FUNCTION_BLOCK StackerCraneProcess
VAR_IN_OUT
	bStart : BOOL;
	bHalt : BOOL;
	bResume : BOOL;
	bStop : BOOL;
	fioOutputs : OUTPUTS;
END_VAR
VAR_INPUT
	fioInputs : INPUTS;
	iAlgo: INT;
	iMode: INT;
	iRackSlot : INT;
END_VAR
VAR_OUTPUT
	sCurrentOperation : STRING;
	iTotalPalletsProcessed : INT;
	iPalletsInRack : INT;
	aSlots : ARRAY[1..54] OF BOOL;

END_VAR
VAR
	bFirstStart : BOOL := TRUE;
	
	iStep : INT := 0;
	bPalletWaiting : BOOL;
	startTrig : R_TRIG;
	stopTrig : R_TRIG;
	resumeTrig : R_TRIG;
	haltTrig : R_TRIG;
	iHaltStep : INT;
	mAlgo : INT;
	mMode : INT;
	i : INT;
	iChosenSlot : INT;
	fill : Fill;
	empty : Empty;
	home : Home;
	iCounter :INT;
	exitTimer : TON;
	infoTimer : TON;
	aFillVerticalPositions : ARRAY[1..54] OF INT := [
		1, 10, 19, 28, 37, 46,
		2, 11, 20, 29, 38, 47,
		3, 12, 21, 30, 39, 48,
		4, 13, 22, 31, 40, 49,
		5, 14, 23, 32, 41, 50,
		6, 15, 24, 33, 42, 51,
		7, 16, 25, 34, 43, 52,
		8, 17, 26, 35, 44, 53,
		9, 18, 27, 36, 45, 54
	];
	
	aEmptyVerticalPositions : ARRAY[1..54] OF INT := [
		54, 45, 36, 27, 18, 9,
		53, 44, 35, 26, 17, 8,
		52, 43, 34, 25, 16, 7,
		51, 42, 33, 24, 15, 6,
		50, 41, 32, 23, 14, 5,
		49, 40, 31, 22, 13, 4,
		48, 39, 30, 21, 12, 3,
		47, 38, 29, 20, 11, 2,
		46, 37, 28, 19, 10, 1
	];
	storedOutputs : OUTPUTS;
	haltedOutputs : OUTPUTS;
	sStoredCurrentOp : STRING;
	
END_VAR

VAR CONSTANT
	AVAILABLE_SLOTS: INT := 54;
END_VAR

startTrig(CLK:=bStart);
stopTrig(CLK:=bStop);
resumeTrig(CLK:=bResume);
haltTrig(CLK:=bHalt);
exitTimer(PT:=T#5S);
infoTimer(PT:=T#5S);

fill(
	fioOutputs:=fioOutputs,
	iPalletsInRack:=iPalletsInRack,
	sCurrentOperation:=sCurrentOperation,
	aSlots:=aSlots,
	fioInputs:=fioInputs,
	bHalt:=haltTrig.Q,
	bResume:=resumeTrig.Q);	
	
empty(
	fioOutputs:=fioOutputs,
	iPalletsInRack:=iPalletsInRack,
	sCurrentOperation:=sCurrentOperation,
	aSlots:=aSlots,
	fioInputs:=fioInputs,
	bHalt:=haltTrig.Q,
	bResume:=resumeTrig.Q);		

home(
	fioOutputs:=fioOutputs,
	iPalletsInRack:=iPalletsInRack,
	sCurrentOperation:=sCurrentOperation,
	aSlots:=aSlots,
	fioInputs:=fioInputs,
	bPalletWaiting:=bPalletWaiting,
	bHalt:=haltTrig.Q,
	bResume:=resumeTrig.Q);	
	
IF startTrig.Q 
	AND iStep = 0
	THEN
	resetInputs();
	mAlgo := iAlgo;
	mMode := iMode;
	IF bFirstStart
		THEN
		bFirstStart := FALSE;
		iStep := 3000;
	ELSE
		iStep := 10;
	END_IF
END_IF

IF startTrig.Q 
	AND iStep = 2000
	THEN
	resetInputs();
	//Home
	iStep := 3000;
END_IF

IF resumeTrig.Q 
	AND iStep  = 1050
	THEN
	resetInputs();
	iStep := 1100;
END_IF

IF haltTrig.Q
	THEN
	resetInputs();
	sStoredCurrentOp := sCurrentOperation;
	sCurrentOperation := 'Halted';
	iHaltStep := iStep;
	iStep := 1000;	
END_IF

IF stopTrig.Q
	THEN
	resetInputs();
	sCurrentOperation := 'Stopped';
	iStep :=  2000;
END_IF

CASE iStep OF
	0:
	 	sCurrentOperation := 'Idle';
		infoTimer.IN := FALSE;
		exitTimer.IN := FALSE;
		resetInputs();

	10: 
		IF mMode = 1 // Fill
			AND iPalletsInRack < 54
			AND NOT (mAlgo = 3 AND aSlots[iRackSlot]) 
			THEN
			iTotalPalletsProcessed := iTotalPalletsProcessed + 1;
			IF bPalletWaiting 
				THEN
				
				sCurrentOperation := 'Pallet already waiting';
			ELSE
				// Emit Pallet		
				fioOutputs.bEmitPallet := TRUE;
				// Start Entry Conveyors
				fioOutputs.bEntryRollerConveyor := TRUE;
				fioOutputs.bEntryLoadingConveyor := TRUE;
				sCurrentOperation := 'Entry Conveyor started';
			END_IF

			iStep := 20;
		ELSIF mMode = 2
			AND iPalletsInRack > 0 // empty
			AND NOT (mAlgo = 3 AND NOT aSlots[iRackSlot]) 
			THEN
			iStep := 60;
			
		ELSE // Not mplemented yet
			iStep := 0;
		END_IF
		
	// ------------------------------------------------------------------------ Fill operation --------------------------------------------------------
	20: // Check Pallet in Loading Conveyor
		IF fioInputs.bEntrySensor
			THEN
			// Stop emitting and stop conveyors
			fioOutputs.bEntryRollerConveyor := FALSE;
			fioOutputs.bEntryLoadingConveyor := FALSE;
			fioOutputs.bEmitPallet := FALSE;	
			iStep := 30;	
		END_IF
		
	30: // Check if space available in rack
		IF iPalletsInRack < AVAILABLE_SLOTS
			THEN
			iStep := 40;
		ELSE
			// Halt operations
			sCurrentOperation := 'No available space in rack';
			infoTimer.IN := TRUE;
			IF infoTimer.Q
				THEN
				infoTimer.IN := FALSE;
				iStep:=0;
			END_IF
			
		END_IF
		
	40: // Check algo for fill operation
	
		IF mAlgo = 1 // Horizontal
			THEN
			sCurrentOperation := 'Filling horizontally';
			FOR i := 1 TO 54 DO
				IF aSlots[i] = FALSE
					THEN
					iChosenSlot := i;
					EXIT;
				END_IF
			END_FOR
			iStep := 50;
		ELSIF mAlgo = 2 // Vertical
			THEN
			sCurrentOperation := 'Filling vertically';
			FOR i := 1 TO 54 DO
				IF aSlots[aFillVerticalPositions[i]] = FALSE
					THEN
					iChosenSlot := aFillVerticalPositions[i];
					EXIT;
				END_IF
			END_FOR
			iStep := 50;	
		ELSIF mAlgo = 3 // Manual
			THEN
			sCurrentOperation := 'Filling manually';
			iChosenSlot := iRackSlot;
			iStep := 50;
		ELSE
			// Halt operations
			iStep := 1000;
		END_IF
		
	50:
		fill.bStart := TRUE;
		fill.iSlotPosition := iChosenSlot;
		bPalletWaiting := FALSE;
		IF fill.bDone THEN
			fill.bStart := FALSE;
			iStep := 0;
		END_IF
		
		
	// ------------------------------------------------------------------------ Empty operation --------------------------------------------------------
	60: //Check algo for empty operation
	
		IF mAlgo = 1 // Horizontal
			THEN
			sCurrentOperation := 'Emptying horizontally';
			iCounter := 54;
			WHILE iCounter<>0 DO
				IF aSlots[iCounter] 
					THEN
					iChosenSlot := iCounter;
					EXIT;
				END_IF
    			iCounter := iCounter-1;
			END_WHILE
			
			iStep := 70;
		ELSIF mAlgo = 2 // Vertical
			THEN
			sCurrentOperation := 'Emptying vertically';
			FOR i := 1 TO 54 DO
				IF aSlots[aEmptyVerticalPositions[i]] 
					THEN
					iChosenSlot := aEmptyVerticalPositions[i];
					EXIT;
				END_IF
			END_FOR
			iStep := 70;
		ELSIF mAlgo = 3 // Manual
			THEN
			sCurrentOperation := 'Emptying manually';
			iChosenSlot := iRackSlot;
			iStep := 70;
		ELSE
			// Halt operations
			iStep := 1000;
		END_IF
		
	70:
		empty.bStart := TRUE;
		empty.iSlotPosition := iChosenSlot;
		IF empty.bDone THEN
			empty.bStart := FALSE;
			iStep := 80;
		END_IF
		
	80:
		fioOutputs.bExitLoadingConveyor := TRUE;
		fioOutputs.bExitRollerConveyor := TRUE;
		IF fioInputs.bExitSensor
			THEN
			iStep := 90;
		END_IF
		
	90:
		exitTimer.IN := TRUE;
		IF exitTimer.Q
			THEN
			exitTimer.IN := FALSE;
			fioOutputs.bExitLoadingConveyor := FALSE;
			fioOutputs.bExitRollerConveyor := FALSE;
			iStep:=0;
		END_IF
		
	1000:
		storedOutputs := fioOutputs;
		haltedOutputs.bSCLeft := fioOutputs.bSCLeft;
		haltedOutputs.bSCRight := fioOutputs.bSCRight;
		haltedOutputs.bSCLift := fioOutputs.bSCLift;
		fioOutputs := haltedOutputs;
		iStep:=1050;
		
	1050:;
	
	1100:
		fioOutputs := storedOutputs;
		sCurrentOperation := sStoredCurrentOp;
		iStep := iHaltStep;	
		
	2000:
		fioOutputs.iSCPosition := 0;
		fill.bStart := FALSE;
		empty.bStart := FALSE;
		fioOutputs.bEntryLoadingConveyor := FALSE;
		fioOutputs.bEntryRollerConveyor := FALSE;
		fioOutputs.bExitLoadingConveyor := FALSE;
		fioOutputs.bExitRollerConveyor := FALSE;
		exitTimer.IN := FALSE;

		resetInputs();	
		
	3000:
	
		home.bStart := TRUE;
		IF home.bDone THEN
			home.bStart := FALSE;
			iStep := 10;
		END_IF
		
END_CASE

METHOD PRIVATE resetInputs : BOOL
VAR_INPUT
END_VAR
bStart := FALSE;
bHalt := FALSE;
bResume := FALSE;
bStop := FALSE;
END_METHOD

END_FUNCTION_BLOCK

(* stored: Version 1.1.0.1, ProductVersion 3.1.4024.10
   POU StackerCraneProcess: Id {b4bd5f7d-e366-4bba-8281-bae6ed04b2d2}, SpecialFunc None
   Method resetInputs: Id {7f98eaa7-e02f-48c5-bb0c-20e0578da105} *)
